FUNCTION_BLOCK Camera (* Basic FB with empty ECC *)
  (* Standard: 61499-2 *)
  (* Version 1.0, 2021-08-03, AK121668 *)
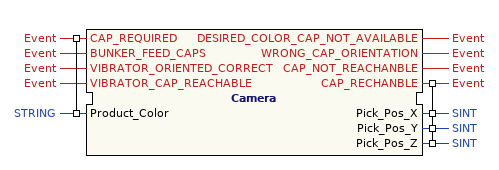
  EVENT_INPUT
    CAP_REQUIRED WITH Product_Color;
    BUNKER_FEED_CAPS;
    VIBRATOR_ORIENTED_CORRECT;
    VIBRATOR_CAP_REACHABLE;
  END_EVENT
  EVENT_OUTPUT
    DESIRED_COLOR_CAP_NOT_AVAILABLE;
    WRONG_CAP_ORIENTATION;
    CAP_NOT_REACHANBLE;
    CAP_RECHANBLE WITH Pick_Pos_X, Pick_Pos_Y, Pick_Pos_Z;
  END_EVENT
  VAR_INPUT
    Product_Color : STRING;
  END_VAR
  VAR_OUTPUT
    Pick_Pos_X : SINT;
    Pick_Pos_Y : SINT;
    Pick_Pos_Z : SINT;
  END_VAR
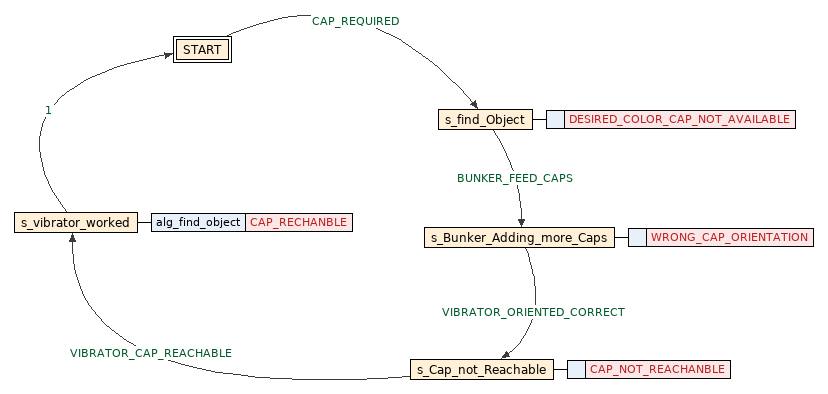
  EC_STATES
    START; (* Initial State *)
    s_find_Object : -> DESIRED_COLOR_CAP_NOT_AVAILABLE;
    s_Bunker_Adding_more_Caps : -> WRONG_CAP_ORIENTATION;
    s_vibrator_worked : alg_find_object -> CAP_RECHANBLE;
    s_Cap_not_Reachable : -> CAP_NOT_REACHANBLE;
  END_STATES
  EC_TRANSITIONS
    START TO s_find_Object := CAP_REQUIRED;
    s_find_Object TO s_Bunker_Adding_more_Caps := BUNKER_FEED_CAPS;
    s_vibrator_worked TO START := 1;
    s_Bunker_Adding_more_Caps TO s_Cap_not_Reachable := VIBRATOR_ORIENTED_CORRECT;
    s_Cap_not_Reachable TO s_vibrator_worked := VIBRATOR_CAP_REACHABLE;
  END_TRANSITIONS
  ALGORITHM alg_find_object IN ST: (* // *)
//
Pick_Pos_X := 100;
Pick_Pos_Y := 50;
Pick_Pos_Z := 5;
  END_ALGORITHM
END_FUNCTION_BLOCK
